FUNCTION_BLOCK T_Cylinder EXTENDS T_NamedBase IMPLEMENTS I_Cylinder
VAR
END_VAR

END_FUNCTION_BLOCK

(* stored: Version 1.1.0.1, ProductVersion 3.1.4024.12
   POU T_Cylinder: Id {d09c98af-cbe5-4c84-9fab-f7b1717b81db}, SpecialFunc None *)
